// TIA Portal V20 export
// export: Created 2025-12-01T14:57:28.1471594Z, ExportSetting None, DisplayName Totally Integrated Automation Portal, DisplayVersion V20 Update 3, DisplayName TIA Portal Openness, DisplayVersion V20 Update 3, DisplayName TIA Portal Version Control Interface, DisplayVersion V20 Update 3, DisplayName STEP 7 Professional, DisplayVersion V20 Update 3, DisplayName STEP 7 Safety, DisplayVersion V20 Update 2, DisplayName WinCC Basic/Comfort/Advanced, DisplayVersion V20 Update 3, DisplayName WinCC Professional, DisplayVersion V20 Update 3, DisplayName WinCC Unified, DisplayVersion V20 Update 3
FUNCTION_BLOCK "FB600_ControlPosicion_Quimarox"   // FB600, LAD
{ S7_Optimized_Access := 'FALSE' }
AUTHOR : Naibes
// stored: AutoNumber false, SetENOAutomatically false
   VAR_INPUT
      ID_Quimarox : UInt;
      Detector_paso_cero : Bool;
      V_Cnt_Tout_paso_Cero : UDInt;
      Dato_encoder : DInt;   // Tiene que ser una entrada del DB de encoders
   END_VAR
   VAR_OUTPUT
      numero_vagon_entrada : Int;
      avance_vagon_entrada : Int;
      avance_total : Int;
   END_VAR
   VAR
      maux_fp_detect_cero : Bool;
      mem_cnt_tout : UDInt;
      total_registros : Int;
   END_VAR
   VAR_TEMP
      contador_elementos : Int;
      pulsos_transcurridos : DInt;
      avance_vagon_ref : DInt;
      num_vag_in : Int;
      Avance_vag_inic : Int;
      aux_int : Int;
      Avance_vagon_X : Int;
      salto : Int;
      basura : Bool;
   END_VAR
BEGIN

NETWORK
TITLE = Variable provisional
//=====================================================================================================================

//=====================================================================================================================

NETWORK
TITLE = 
// Control de posicionamiento y memorias de encoder

      CALL  "FC600_ini+ref_dato_encoder_NEW"
      ( Detector_referencia := #Detector_paso_cero,
        ID_Quimarox         := #ID_Quimarox,
        dato_encoder_actual := #Dato_encoder,
        V_cnt_tout_refresco := #V_Cnt_Tout_paso_Cero,
        m_aux_pf_detect     := #maux_fp_detect_cero,
        MEM_CNT_TOUT        := #mem_cnt_tout
      );


NETWORK
TITLE = Variable provisional
      SET;
      A     "DB600_ConfigQuimarox".Quimarox[#ID_Quimarox].datos_config.DatosTrabajo.Error_Referenciacion;  // #Error_Referenciacion
      R     "DB600_ConfigQuimarox".Quimarox[#ID_Quimarox].datos_config.DatosTrabajo.Memoria_Inicializacion;  //#Mem_Inicializacion

NETWORK
TITLE = Borrado de DB Posiciones asociadas a elementos
// aqui se borran todas las posiciones asociadas a los elementos para luego 
// posteriormente cargar los datos que correspondan. Esto lo hacemos antes de 
// comprobar si está inicializado o no para que si perdemos la referencia dejemos 
// de tener datos.
//=====================================================================================================================

      L     1;  //Iniciamos Cont. Bytes a Borrar     Cuidado con los temporales, inicializar siempre
      T     #contador_elementos;


bucl: NOP   0;
//=====================================================================================================================
//limpia los datos antes de calcular los nuevos

      SET;
      R     "DB602_ElementosQuimarox".Quimarox[#ID_Quimarox].Elementos[#contador_elementos].Hay_Carrier_en_ventana;  //Vagon_en_Ventana
      L     0;
      T     "DB602_ElementosQuimarox".Quimarox[#ID_Quimarox].Elementos[#contador_elementos].Numero_carrier;  //Vagon_Asociado
      T     "DB602_ElementosQuimarox".Quimarox[#ID_Quimarox].Elementos[#contador_elementos].Avance_carrier;  //Posicion_Vagon


      L     #contador_elementos;
      L     "CTE_MaxNumElementos";
      >=I;
      JC    cont;

      L     1;
      L     #contador_elementos;
      +I;
      T     #contador_elementos;

      JU    bucl;
//=====================================================================================================================

NETWORK
TITLE = 
//=====================================================================================================================

cont: AN    "DB600_ConfigQuimarox".Quimarox[#ID_Quimarox].datos_config.DatosTrabajo.Memoria_Inicializacion;
      JC    fin1;  //el primer vagon y no podemos calcular nada

//=====================================================================================================================

NETWORK
TITLE = 
// con el dato del encoder de referencia del primer vagon calculamos el elemento 
// que se encuentra en la entrada del sorter para utilizarlo de vagon de referencia
//===================================================================================================
//aqui comprobaremos si ha pasado por el máximo o no y en funcion de eso calcularemos el numero
//de pulsos que han transcurrido desde la referenciación del primer vagon
//====================================================================================================

      L     "DB600_ConfigQuimarox".Quimarox[#ID_Quimarox].datos_config.DatosTrabajo.Memoria_Dato_Encoder;  //#Mem_Dato_Encoder
      L     #Dato_encoder;
      >D;
      JCN   MEN;

      L     "DB600_ConfigQuimarox".Quimarox[#ID_Quimarox].datos_config.maximo_encoder;
      L     "DB600_ConfigQuimarox".Quimarox[#ID_Quimarox].datos_config.DatosTrabajo.Memoria_Dato_Encoder;
      -D;
      L     #Dato_encoder;
      +D;
      T     #pulsos_transcurridos;
      JU    CLC;

//=====================================================================================================================

MEN:  L     #Dato_encoder;
      L     "DB600_ConfigQuimarox".Quimarox[#ID_Quimarox].datos_config.DatosTrabajo.Memoria_Dato_Encoder;
      -D;
      T     #pulsos_transcurridos;


//============================================================================================================================================
// NIEVES: Calculo del avance del vagón de referencia

CLC:  L     #pulsos_transcurridos;
      DTR;
      L     "DB600_ConfigQuimarox".Quimarox[#ID_Quimarox].datos_config.relacion_mm_pulso;  // #Datos_config.relacion_mm_pulso
      *R;
      RND+;
      L     "DB600_ConfigQuimarox".Quimarox[#ID_Quimarox].datos_config.dist_ini_vag_a_phs_mm;  //distancia del punto de deteccion de referencia al punto de referencia 0
      ITD;
      +D;
      T     #avance_vagon_ref;  //en mm

//=====================================================================================================================

//con el dato del avance del vagon de referencia calculamos cual es el vagon que esta en el inicio del sorter
//y cuando ha avanzado respecto del punto de referencia para con este dato calcular la posicion del resto


NETWORK
TITLE = Calculo de posicón del primer vagón
// en funcion del avance del primer vagon calculamos cual es el vagon que se 
// encuentra en el inicio del sorter y cuanto ha avanzado desde el punto de 
// referencia
//=====================================================================================================================
//si no hace bien lo del numero de vagon revisar este punto
      L     #avance_vagon_ref;
      L     "DB600_ConfigQuimarox".Quimarox[#ID_Quimarox].datos_config.Long_Vagon_mm;
      ITD;
      /D;
      L     1;
      +D;
      DTB;
      BTI;
      T     #num_vag_in;  //Calcula y guarda Vagon en posición inicial

      L     #num_vag_in;
      L     "DB600_ConfigQuimarox".Quimarox[#ID_Quimarox].datos_config.Numero_vagones;

      <=I;
      JC    p_1;

//=====================================================================================================================

      L     #num_vag_in;
      L     "DB600_ConfigQuimarox".Quimarox[#ID_Quimarox].datos_config.Numero_vagones;
      -I;
      T     #numero_vagon_entrada;
      JU    p_2;

//=====================================================================================================================
p_1:  L     #num_vag_in;
      T     #numero_vagon_entrada;

//=====================================================================================================================
p_2:  L     #avance_vagon_ref;
      L     "DB600_ConfigQuimarox".Quimarox[#ID_Quimarox].datos_config.Long_Vagon_mm;
      MOD;
      T     #avance_vagon_entrada;
      T     #Avance_vag_inic;  //Calcula y guarda avance Vagon actual en posición inicial

      L     #pulsos_transcurridos;  // Calcula el avance total desde origen
      DTR;
      L     "DB600_ConfigQuimarox".Quimarox[#ID_Quimarox].datos_config.relacion_mm_pulso;
      *R;
      RND+;
      T     #avance_total;

//=====================================================================================================================

NETWORK
TITLE = calculo posicon vagon todos elementos
// aqui vamos realizando los saltos a cada uno de los elementos, calculamos lo que 
// ha avanzado el vagon y si entra dentro de los limites establecidos para dicho 
// elemento cargamos el numero de vagon correspondiente en la posicion asociada a 
// dicho elemento
//===================================================================================================================================

      L     1;
      T     #contador_elementos;

//=====================================================================================================================
//aqui el calculo de lo que ha avanzado el vagon para dicho elemento
//NIEVES


sige: NOP   0;

//=====================================================================================================================

      L     "DB602_ElementosQuimarox".Quimarox[#ID_Quimarox].Elementos[#contador_elementos].posicion_real_elemento;  //#datos_elemento_actual.posicion_real_elemento
      TRUNC;
      L     "DB600_ConfigQuimarox".Quimarox[#ID_Quimarox].datos_config.Long_Vagon_mm;
      ITD;
      MOD;
      T     #aux_int;
      L     "DB600_ConfigQuimarox".Quimarox[#ID_Quimarox].datos_config.Long_Vagon_mm;
      L     #aux_int;
      -I;  //Avance del vagon para el elemento tratado
      L     #Avance_vag_inic;
      +I;
      L     "DB600_ConfigQuimarox".Quimarox[#ID_Quimarox].datos_config.Long_Vagon_mm;
      MOD;
      T     #Avance_vagon_X;

//=====================================================================================================================

NETWORK
TITLE = comparación de la ventana del elemento segun grado de avance
// aqui la comparacion primero con el rango inferior y luego con el rango superior
//=====================================================================================================================
      CLR;
      =     "DB602_ElementosQuimarox".Quimarox[#ID_Quimarox].Elementos[#contador_elementos].Hay_Carrier_en_ventana;  //Inicio Validación elemento en rango Ventana


      L     "DB602_ElementosQuimarox".Quimarox[#ID_Quimarox].Elementos[#contador_elementos].ventana_minima;
      L     #Avance_vagon_X;
      >I;
      JC    vent;

//=====================================================================================================================

      L     "DB602_ElementosQuimarox".Quimarox[#ID_Quimarox].Elementos[#contador_elementos].ventana_maxima;  //apunta a la posicion maxima
      L     #Avance_vagon_X;
      <I;
      JC    vent;

      SET;
      =     "DB602_ElementosQuimarox".Quimarox[#ID_Quimarox].Elementos[#contador_elementos].Hay_Carrier_en_ventana;

//=====================================================================================================================




NETWORK
TITLE = calcular el número de vagón que corresponde
// aqui si se cumple que esta entre los dos rangos, calculamos el numero de vagon 
// que corresponde y lo cargamos en la correspondiente posicion asociada
// 
// al finalizar comprobar que no estamos en el ultimo elemento, si lo estamos, 
// saltar al final, y si no lo estamos pasa al siguiente elemento y spa sige
//=====================================================================================================================
//aqui calculamos el vagon que esta en frente del elemento
// para poder hacer el redondeo tenemos que hacer todo el cálculo en real

vent: L     "DB602_ElementosQuimarox".Quimarox[#ID_Quimarox].Elementos[#contador_elementos].posicion_real_elemento;
      L     #Avance_vag_inic;
      ITD;
      DTR;
      -R;
      L     "DB600_ConfigQuimarox".Quimarox[#ID_Quimarox].datos_config.Long_Vagon_mm;
      ITD;
      DTR;
      /R;
      RND+;
      T     #salto;
      L     #num_vag_in;
      L     #salto;
      -I;
      T     #aux_int;

      L     #aux_int;
      L     1;
      <I;
      JCN   p_3;


//=====================================================================================================================
      L     #aux_int;
      L     "DB600_ConfigQuimarox".Quimarox[#ID_Quimarox].datos_config.Numero_vagones;
      +I;
      T     #aux_int;


//=====================================================================================================================
p_3:  L     #aux_int;
      L     "DB600_ConfigQuimarox".Quimarox[#ID_Quimarox].datos_config.Numero_vagones;
      >I;
      JCN   carg;

      L     #aux_int;
      L     "DB600_ConfigQuimarox".Quimarox[#ID_Quimarox].datos_config.Numero_vagones;
      -I;
      T     #aux_int;

//=====================================================================================================================
carg: L     #aux_int;
      T     "DB602_ElementosQuimarox".Quimarox[#ID_Quimarox].Elementos[#contador_elementos].Numero_carrier;

      L     #Avance_vagon_X;
      T     "DB602_ElementosQuimarox".Quimarox[#ID_Quimarox].Elementos[#contador_elementos].Avance_carrier;

//=====================================================================================================================

      L     #contador_elementos;
      L     "CTE_MaxNumElementos";
      ==I;
      JC    fin;

      L     #contador_elementos;
      L     1;
      +I;
      T     #contador_elementos;

      JU    sige;

//=====================================================================================================================

NETWORK
TITLE = 
//=====================================================================================================================
fin:  BE;


//=====================================================================================================================
fin1: L     0;
      T     #numero_vagon_entrada;
      T     #avance_vagon_entrada;


//=====================================================================================================================
END_FUNCTION_BLOCK
